PROGRAM UpdateSek
VAR
	SekUpdate_R1			:FB_UpdateSek;
	SekUpdate_R2			:FB_UpdateSek;
	SekUpdate_R3			:FB_UpdateSek;
	SekUpdate_R4			:FB_UpdateSek;
	SekUpdate_R5			:FB_UpdateSek;
	SekUpdate_R6			:FB_UpdateSek;
	SekUpdate_R7			:FB_UpdateSek;
END_VAR

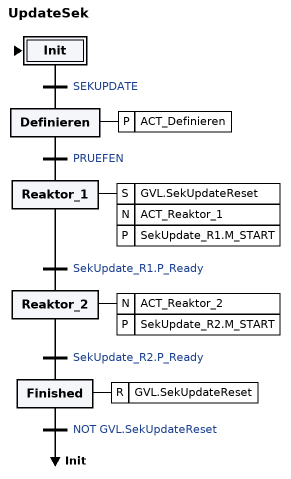
INITIAL_STEP Init:
END_STEP
TRANSITION FROM Init TO Definieren
    := SEKUPDATE;
END_TRANSITION
STEP Definieren:
    ACT_Definieren(P);
END_STEP
TRANSITION FROM Definieren TO Reaktor_1
    := PRUEFEN;
END_TRANSITION
STEP Reaktor_1:
    GVL.SekUpdateReset(S);
    ACT_Reaktor_1(N);
    SekUpdate_R1.M_START(P);
END_STEP
TRANSITION FROM Reaktor_1 TO Reaktor_2
    := SekUpdate_R1.P_Ready;
END_TRANSITION
STEP Reaktor_2:
    ACT_Reaktor_2(N);
    SekUpdate_R2.M_START(P);
END_STEP
TRANSITION FROM Reaktor_2 TO Finished
    := SekUpdate_R2.P_Ready;
END_TRANSITION
STEP Finished:
    GVL.SekUpdateReset(R);
END_STEP
TRANSITION FROM Finished TO Init
    := NOT GVL.SekUpdateReset;
END_TRANSITION

ACTION ACT_Definieren:
IF GVL.SekUpdate_1 THEN
	CASE GVL.R1_CW.SekReakt OF
		1:	GVL.SekControlWord.R1 := TRUE;
		2:	GVL.SekControlWord.R2 := TRUE;
		3:	GVL.SekControlWord.R3 := TRUE;
		4:	GVL.SekControlWord.R4 := TRUE;
		5:	GVL.SekControlWord.R5 := TRUE;
		6:	GVL.SekControlWord.R6 := TRUE;
		7:	GVL.SekControlWord.R7 := TRUE;
	END_CASE
END_IF

IF GVL.SekUpdate_2 THEN
	CASE GVL.R2_CW.SekReakt OF
		1:	GVL.SekControlWord.R1 := TRUE;
		2:	GVL.SekControlWord.R2 := TRUE;
		3:	GVL.SekControlWord.R3 := TRUE;
		4:	GVL.SekControlWord.R4 := TRUE;
		5:	GVL.SekControlWord.R5 := TRUE;
		6:	GVL.SekControlWord.R6 := TRUE;
		7:	GVL.SekControlWord.R7 := TRUE;
	END_CASE
END_IF

IF GVL.SekUpdate_3 THEN
	CASE GVL.R3_CW.SekReakt OF
		1:	GVL.SekControlWord.R1 := TRUE;
		2:	GVL.SekControlWord.R2 := TRUE;
		3:	GVL.SekControlWord.R3 := TRUE;
		4:	GVL.SekControlWord.R4 := TRUE;
		5:	GVL.SekControlWord.R5 := TRUE;
		6:	GVL.SekControlWord.R6 := TRUE;
		7:	GVL.SekControlWord.R7 := TRUE;
	END_CASE
END_IF

IF GVL.SekUpdate_4 THEN
	CASE GVL.R4_CW.SekReakt OF
		1:	GVL.SekControlWord.R1 := TRUE;
		2:	GVL.SekControlWord.R2 := TRUE;
		3:	GVL.SekControlWord.R3 := TRUE;
		4:	GVL.SekControlWord.R4 := TRUE;
		5:	GVL.SekControlWord.R5 := TRUE;
		6:	GVL.SekControlWord.R6 := TRUE;
		7:	GVL.SekControlWord.R7 := TRUE;
	END_CASE
END_IF

IF GVL.SekUpdate_5 THEN
	CASE GVL.R5_CW.SekReakt OF
		1:	GVL.SekControlWord.R1 := TRUE;
		2:	GVL.SekControlWord.R2 := TRUE;
		3:	GVL.SekControlWord.R3 := TRUE;
		4:	GVL.SekControlWord.R4 := TRUE;
		5:	GVL.SekControlWord.R5 := TRUE;
		6:	GVL.SekControlWord.R6 := TRUE;
		7:	GVL.SekControlWord.R7 := TRUE;
	END_CASE
END_IF

IF GVL.SekUpdate_6 THEN
	CASE GVL.R6_CW.SekReakt OF
		1:	GVL.SekControlWord.R1 := TRUE;
		2:	GVL.SekControlWord.R2 := TRUE;
		3:	GVL.SekControlWord.R3 := TRUE;
		4:	GVL.SekControlWord.R4 := TRUE;
		5:	GVL.SekControlWord.R5 := TRUE;
		6:	GVL.SekControlWord.R6 := TRUE;
		7:	GVL.SekControlWord.R7 := TRUE;
	END_CASE
END_IF

IF GVL.SekUpdate_7 THEN
	CASE GVL.R7_CW.SekReakt OF
		1:	GVL.SekControlWord.R1 := TRUE;
		2:	GVL.SekControlWord.R2 := TRUE;
		3:	GVL.SekControlWord.R3 := TRUE;
		4:	GVL.SekControlWord.R4 := TRUE;
		5:	GVL.SekControlWord.R5 := TRUE;
		6:	GVL.SekControlWord.R6 := TRUE;
		7:	GVL.SekControlWord.R7 := TRUE;
	END_CASE
END_IF
END_ACTION

ACTION ACT_Reaktor_1:
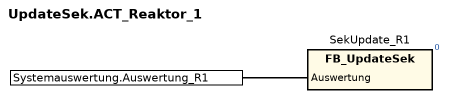
SekUpdate_R1(Auswertung := Systemauswertung.Auswertung_R1); // FB_UpdateSek
END_ACTION

ACTION ACT_Reaktor_2:
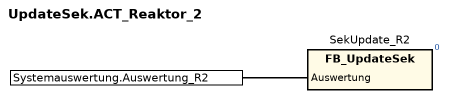
SekUpdate_R2(Auswertung := Systemauswertung.Auswertung_R2); // FB_UpdateSek
END_ACTION

TRANSITION PRUEFEN:
IF GVL.SekControlWord.R1 OR GVL.SekControlWord.R2 OR GVL.SekControlWord.R3 OR GVL.SekControlWord.R4 OR GVL.SekControlWord.R5 OR GVL.SekControlWord.R6 OR GVL.SekControlWord.R7 THEN
	PRUEFEN := TRUE;
ELSE 
	PRUEFEN := FALSE;
END_IF
END_TRANSITION

TRANSITION SEKUPDATE:
IF GVL.SekUpdate_1 OR
	GVL.SekUpdate_2 OR
	GVL.SekUpdate_3 OR
	GVL.SekUpdate_4 OR
	GVL.SekUpdate_5 OR
	GVL.SekUpdate_6 OR
	GVL.SekUpdate_7 THEN
	
	SEKUPDATE := TRUE;
ELSE 
	SEKUPDATE := FALSE;
END_IF
END_TRANSITION

END_PROGRAM

(* stored: Version 1.1.0.1, ProductVersion 3.1.4024.12
   POU UpdateSek: Id {d2f2f3d7-860e-4d1f-b76c-f35ecca23e52}, SpecialFunc None
   Folder 01_Aktionen: Id {b1f02134-4736-477c-b46b-295dfb9f8888}
   Folder 02_Transitionen: Id {0ce38f20-8f8d-48ca-b870-0d39b92feb68}
   Action ACT_Definieren: Id {adec9976-4b37-4752-b6de-1aa0a6dd0fc1}
   Action ACT_Reaktor_1: Id {ad590887-0c4d-44df-a20c-3161d22c739d}
   Action ACT_Reaktor_2: Id {055f6b88-5b2f-4078-8de6-2b0f76e95dc2}
   Transition PRUEFEN: Id {a686afab-275f-4f45-b7ea-0cb39f839168}
   Transition SEKUPDATE: Id {2b8ada42-f7c2-4dc9-8c93-6579116d034c} *)
